Staubli VAL3: OnF3.pgx

program OnF3()
  local string l_sYesNo[2]
  local num l_i
begin
  //删除
  l_sYesNo[0]="是"
  l_sYesNo[1]="否"
  call user:questionDialog("是否删除此路径?",l_sYesNo,l_i)
  if l_i==0 or l_i==1
    if sFileList[nSelected]!=""
      libDelete(sFolder+sFileList[nSelected])
      delete(sFileList[nSelected])
      bListRefresh=true
    endIf
  endIf
  bUserRefresh=true

end
